PROGRAM MAIN
VAR
	m : INT;
END_VAR

m := m + 1;
PrgMqttCom();

END_PROGRAM

(* stored: Version 1.1.0.1, ProductVersion 3.1.4024.5
   POU MAIN: Id {e4c4f930-8f79-4895-a54f-5256381f76bd}, SpecialFunc None *)
